PROGRAM Q1
VAR
	loop : INT := 1;
END_VAR

END_PROGRAM

(* stored: Version 1.1.0.1, ProductVersion 3.1.4024.12
   POU Q1: Id {9b20c000-40aa-4785-aadb-ca6e9635d130}, SpecialFunc None *)
